// TIA Portal project "SolarInverterDemo" (V15.1)

(* hardware
DEVICE "S7-1200 station_1"  S7-1200 Station
   slot 0: "Rack_0"  S7-1200 Rack  Rack  V1.0
   slot 1: "PLC_1"  CPU 1214C DC/DC/DC  6ES7 214-1AG40-0XB0  V4.3
*)

// ===== PLC "PLC_1"  CPU 1214C DC/DC/DC =====

DATA_BLOCK "MB_HoldingReg"   // DB1
{ S7_Optimized_Access := 'FALSE' }
VERSION : 0.1
// ============================================================================
//   ModbusManager Pro - Siemens S7-1200 demo
//   Solar inverter simulation exposed over Modbus TCP (MB_SERVER)
// 
//   Import:  TIA Portal -> External source files -> Add new external file
//            -> select this .scl -> right-click -> "Generate blocks from source"
//   Then:    call "SolarInverterDemo" cyclically in OB1 (see README).
// 
//   Holding register map (0-based Modbus addresses): see README.
//   Word order for 32-bit values: BIG-ENDIAN (high word at lower address).
//  ============================================================================
//  ---------------------------------------------------------------------------
//   Holding-register data block.
//   MUST be NON-optimized access so MB_HOLD_REG resolves to a contiguous area.
//  ---------------------------------------------------------------------------
   VAR
      Reg : Array[0..49] of Word;   // 50 words of headroom; 0..11 used
   END_VAR
BEGIN
END_DATA_BLOCK

DATA_BLOCK "SolarInverterDemo_DB"   // DB2
{ S7_Optimized_Access := 'TRUE' }
VERSION : 0.1
// stored: InstanceOfName SolarInverterDemo
"SolarInverterDemo"
BEGIN
END_DATA_BLOCK

FUNCTION_BLOCK "SolarInverterDemo"   // FB1, SCL
{ S7_Optimized_Access := 'TRUE' }
VERSION : 0.1
// ---------------------------------------------------------------------------
//   Simulation + Modbus TCP server
//  ---------------------------------------------------------------------------
   VAR_INPUT
      Enable : Bool := TRUE;
   END_VAR
   VAR
      instMbServer : MB_SERVER;   // multi-instance Modbus TCP server
      angle : Real := 0.0;   // sun angle: 0..PI = sunrise..sunset
      powerKW : Real;
      dcVoltage : Real;
      dcCurrent : Real;
      string1A : Real;
      gridFreq : Real;
      invTemp : Real;
      soc : Real := 50.0;   // battery state-of-charge %
      dayEnergy : Real := 0.0;   // kWh today
      totalEnergy : Real := 0.0;   // kWh lifetime
      statusWord : Word;
      tmpDI : DInt;
      tmpDW : DWord;
      connSettings : TCON_IP_v4;   // Modbus TCP connection (passive server)
      initDone : Bool := FALSE;
      cycleTimer : TON_TIME;   // paces the simulation independent of scan time
   END_VAR
BEGIN

   // ===== Simulation pacing: advance one step every 50 ms ========
   // Decouples demo speed from PLC scan time -> smooth, ~16 s "day".
   #cycleTimer(IN := NOT #cycleTimer.Q,
               PT := T#50MS);

   IF #Enable AND #cycleTimer.Q THEN

       // ===== Day-cycle angle =====================================
       // Larger step = faster day. 0.01/scan gives a ~30 s demo "day".
       #angle := #angle + 0.01;
       IF #angle > 3.14159 THEN
           #angle := -1.0;        // negative = night (power clamps to 0)
           #dayEnergy := 0.0;         // reset daily yield at new day
       END_IF;

       // ===== Simulated process values ============================
       #powerKW := 50.0 * SIN(#angle);            // solar bell curve, 0..50 kW
       IF #powerKW < 0.0 THEN
           #powerKW := 0.0;
       END_IF;

       #dcVoltage := 620.0 + 30.0 * SIN(#angle);  // ~590..650 V

       IF #powerKW > 0.5 THEN
           #dcCurrent := (#powerKW * 1000.0) / #dcVoltage;   // I = P / U
       ELSE
           #dcCurrent := 0.0;
       END_IF;
       #string1A := #dcCurrent * 0.5;             // one of two PV strings

       #gridFreq := 50.0 + 0.05 * SIN(#angle * 6.0);        // ~49.95..50.05 Hz
       #invTemp := 25.0 + #powerKW * 0.6;                  // 25..55 deg C

       // Battery SOC: charges in sun, drains at night
       IF #powerKW > 10.0 THEN
           #soc := #soc + 0.05;
       ELSE
           #soc := #soc - 0.03;
       END_IF;
       IF #soc > 100.0 THEN
           #soc := 100.0;
       END_IF;
       IF #soc < 0.0 THEN
           #soc := 0.0;
       END_IF;

       // Energy accumulation (demo factor - tune to taste)
       #dayEnergy := #dayEnergy + #powerKW * 0.015;
       #totalEnergy := #totalEnergy + #powerKW * 0.015;

       // ===== Status word (bitfield) ==============================
       #statusWord := 0;
       IF #powerKW > 0.5 THEN
           #statusWord := #statusWord OR 16#0001;
       END_IF; // bit0 grid-connected
       IF #invTemp > 52.0 THEN
           #statusWord := #statusWord OR 16#0004;
       END_IF; // bit2 derating
       IF #powerKW <= 0.5 THEN
           #statusWord := #statusWord OR 16#0008;
       END_IF; // bit3 standby/night
       // bit1 (fault) stays 0 in normal demo

       // ===== Write to holding registers (0-based addresses) ======
       "MB_HoldingReg".Reg[0] := INT_TO_WORD(REAL_TO_INT(#powerKW * 10.0));  // 40001 AC power  x10  kW
       "MB_HoldingReg".Reg[1] := INT_TO_WORD(REAL_TO_INT(#dcVoltage));  // 40002 DC volts  x1   V
       "MB_HoldingReg".Reg[2] := INT_TO_WORD(REAL_TO_INT(#dcCurrent * 10.0));  // 40003 DC amps   x10  A
       "MB_HoldingReg".Reg[3] := INT_TO_WORD(REAL_TO_INT(#gridFreq * 100.0)); // 40004 frequency x100 Hz
       "MB_HoldingReg".Reg[4] := INT_TO_WORD(REAL_TO_INT(#invTemp * 10.0));  // 40005 temp      x10  deg C

       // 40006/40007 daily energy, U32 x100 kWh, hi word first
       #tmpDI := REAL_TO_DINT(#dayEnergy * 100.0);
       #tmpDW := DINT_TO_DWORD(#tmpDI);
       "MB_HoldingReg".Reg[5] := DWORD_TO_WORD(SHR(IN := #tmpDW, N := 16));    // hi
       "MB_HoldingReg".Reg[6] := DWORD_TO_WORD(#tmpDW AND 16#0000FFFF);        // lo

       // 40008/40009 total energy, U32 x1 kWh, hi word first
       #tmpDI := REAL_TO_DINT(#totalEnergy);
       #tmpDW := DINT_TO_DWORD(#tmpDI);
       "MB_HoldingReg".Reg[7] := DWORD_TO_WORD(SHR(IN := #tmpDW, N := 16));    // hi
       "MB_HoldingReg".Reg[8] := DWORD_TO_WORD(#tmpDW AND 16#0000FFFF);        // lo

       "MB_HoldingReg".Reg[9] := INT_TO_WORD(REAL_TO_INT(#string1A * 10.0));  // 40010 string 1 x10 A
       "MB_HoldingReg".Reg[10] := INT_TO_WORD(REAL_TO_INT(#soc));  // 40011 SOC      x1  %
       "MB_HoldingReg".Reg[11] := #statusWord;                                // 40012 status bitfield

   END_IF;

   // ===== Modbus TCP connection settings (set once) ===============
   // Passive TCP server on port 502, accepts any client.
   IF NOT #initDone THEN
       #connSettings.InterfaceId := 64;          // HW id of PROFINET interface - VERIFY (System constants, often 64 or 100)
       #connSettings.ID := 1;                     // unique connection id (1..4095)
       #connSettings.ConnectionType := 16#0B;     // 11 = TCP
       #connSettings.ActiveEstablished := FALSE;  // FALSE = passive server (waits for client)
       #connSettings.RemoteAddress.ADDR[1] := 0;  // 0.0.0.0 = accept any client
       #connSettings.RemoteAddress.ADDR[2] := 0;
       #connSettings.RemoteAddress.ADDR[3] := 0;
       #connSettings.RemoteAddress.ADDR[4] := 0;
       #connSettings.RemotePort := 0;             // 0 for server
       #connSettings.LocalPort := 502;            // Modbus TCP port
       #initDone := TRUE;
   END_IF;

   // ===== Modbus TCP server - call every scan =====================
   #instMbServer(DISCONNECT := FALSE,
                 CONNECT := #connSettings,
                 MB_HOLD_REG := "MB_HoldingReg".Reg);
END_FUNCTION_BLOCK

ORGANIZATION_BLOCK "Main"   // OB1, LAD, ProgramCycle
TITLE = "Main Program Sweep (Cycle)"
{ S7_Optimized_Access := 'TRUE' }
VERSION : 0.1
   VAR_INPUT
      Initial_Call : Bool;   // Initial call of this OB
      Remanence : Bool;   // =True, if remanent data are available
   END_VAR
BEGIN

REGION Network 1
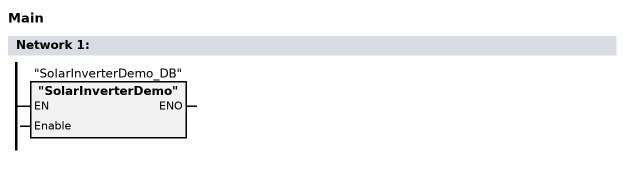
   RUNG wire#powerrail
      "SolarInverterDemo_DB"(Enable :=)
   END_RUNG
   // the same network as SCL:
   "SolarInverterDemo_DB"();   // "SolarInverterDemo"
END_REGION
END_ORGANIZATION_BLOCK